FUNCTION_BLOCK POU EXTENDS fbEM
VAR_INPUT
END_VAR
VAR_OUTPUT
END_VAR
VAR
END_VAR

END_FUNCTION_BLOCK

(* stored: Version 1.1.0.1, ProductVersion 3.1.4024.12
   POU POU: Id {5c7e5af1-d6a9-4457-9412-da2f08e05228}, SpecialFunc None *)
